// TIA Portal V20 export
TYPE "typeCmHmiInterfaceBrakeTest"
// stored: Access Published, Namespace Unit1.Em5
   STRUCT
      transferPnPLeftAxisZ : "LER_typeBrakeTestEmInterface";
      transferPnPRightAxisZ : "LER_typeBrakeTestEmInterface";
   END_STRUCT;
END_TYPE
